// TIA Portal V16 export
// export: Created 2021-06-27T08:23:18.4598635Z, ExportSetting WithDefaults, DisplayName Totally Integrated Automation Portal, DisplayVersion V16 Update 4, DisplayName TIA Portal Version Control Interface, DisplayVersion V16 Update 2, DisplayName TIA Portal Openness, DisplayVersion V16 Update 4, DisplayName STEP 7 Professional, DisplayVersion V16 Update 4, DisplayName STEP 7 Safety, DisplayVersion V16, DisplayName WinCC Advanced, DisplayVersion V16 Update 4
FUNCTION "RunSensors" : Void   // FC8, F_FBD
{ S7_Optimized_Access := 'TRUE' }
VERSION : 0.1
// stored: AutoNumber true, IsIECCheckEnabled false, UDAEnableTagReadback false
   VAR_INPUT
      command_a : "SensorCommand";
      command_b : "SensorCommand";
   END_VAR
   VAR_OUTPUT
      all_ok : Bool;
      last_command_a : "SensorCommand";
   END_VAR
   VAR_TEMP
      a_ok : Bool;
      b_ok : Bool;
   END_VAR
BEGIN

REGION Network 1
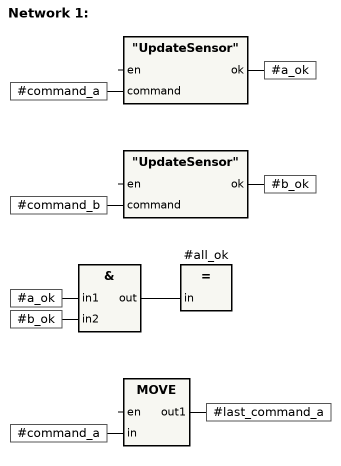
   "UpdateSensor"(command := #command_a, ok => #a_ok);
   "UpdateSensor"(command := #command_b, ok => #b_ok);
   #all_ok := #a_ok AND #b_ok;
   #last_command_a := #command_a;
END_REGION
END_FUNCTION
